(* Logix 5000 project; controller KTC_ball1 vendor 1 type 14 code 149 rev 30.11; software revision 30.00 *)

TASK MainTask (continuous, watchdog 500 ms) : MainProgram

MODULES
   Local : vendor 1 type 14 code 149 (Compact 0, rev 30.11)
      Discrete_IO : Embedded (Compact 1, rev 3.1, Output RPI 20 ms)
END_MODULES

PROGRAM MainProgram   (* main routine MainRoutine *)
VAR
   B3_1 : BOOL;   // gate 3
   pb1 : ALIAS FOR Local:1:I.Data.5;   // ball in gravity shoot
   pb2 : ALIAS FOR Local:1:I.Data.2;   // capacitive sensor
   pb3 : ALIAS FOR Local:1:I.Data.3;   // optical sensor
   pb4 : ALIAS FOR Local:1:I.Data.4;   // inductive sensor
   sol1 : ALIAS FOR Local:1:O.Data.0;   // eject piston valve
   sol2 : ALIAS FOR Local:1:O.Data.1;   // gate1
   sol3 : ALIAS FOR Local:1:O.Data.2;   // gate 2
END_VAR

ROUTINE MainRoutine   (* ladder *)
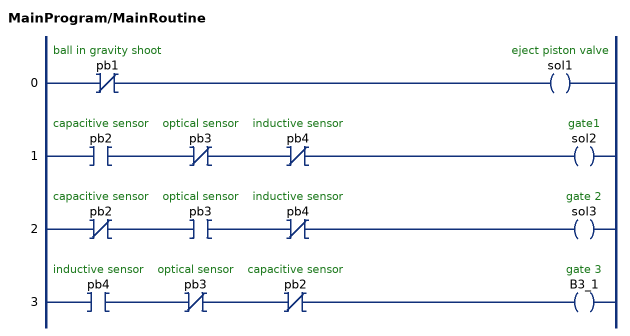
   0: XIO(pb1)OTE(sol1);
   1: XIC(pb2)XIO(pb3)XIO(pb4)OTE(sol2);
   2: XIO(pb2)XIC(pb3)XIO(pb4)OTE(sol3);
   3: XIC(pb4)XIO(pb3)XIO(pb2)OTE(B3_1);
END_ROUTINE
END_PROGRAM
